KUKA KRL program: UnStackPick02.src, UnStackPick02.dat

--- UnStackPick02.src ---
&ACCESS RVP
&COMMENT UnStack Pick02
&REL 35
&PARAM EDITMASK = *
&PARAM TEMPLATE = C:\KRC\Roboter\Template\vorgabe
&PARAM DISKPATH = KRC:\R1\Program\SbtComm010Stack
DEF UnStackPick02( )
;FOLD INI;%{PE}
  ;FOLD BASISTECH INI
    GLOBAL INTERRUPT DECL 3 WHEN $STOPMESS==TRUE DO IR_STOPM ( )
    INTERRUPT ON 3
    BAS (#INITMOV,0 )
  ;ENDFOLD (BASISTECH INI)
  ;FOLD USER INI
    ;Make your modifications here

  ;ENDFOLD (USER INI)
;ENDFOLD (INI)
;FOLD COPY DATA
XPickPos = Comm010CopyTable.PickPos
;ENDFOLD
;FOLD Basic.Frame OUT Frame Dir: PickPosOfsUp, IN x: 0, IN y: 0, IN z: -150, IN a: 0 deg, IN b: 0 deg, IN c: 0 deg ;%{PE}
PickPosOfsUp = set_frame_(0, 0, -150, 0, 0, 0)
;ENDFOLD
;FOLD Basic.Frame OUT Frame Dir: PickPosOfsRUp, IN x: 0, IN y: 0, IN z: -150, IN a: 0 deg, IN b: 0 deg, IN c: 0 deg ;%{PE}
PickPosOfsRUp = set_frame_(0, 0, -150, 0, 0, 0)
;ENDFOLD
;FOLD Basic.ToolOffset IN Source Point Dir: PickPos, IN Offs Dir: PickPosOfsUp, OUT Offset Point Dir: PickPosUp ;%{PE}
XPickPosUp = tool_offs_byframe_(XPickPos, PickPosOfsUp)
;ENDFOLD
;FOLD Basic.ToolOffset IN Source Point Dir: PickPos, IN Offs Dir: PickPosOfsRUp, OUT Offset Point Dir: PickPosRUp ;%{PE}
XPickPosRUp = tool_offs_byframe_(XPickPos, PickPosOfsRUp)
;ENDFOLD
;FOLD SLIN PickPosUp CONT Vel=2 m/s CPDAT1 Tool[1] Base[0] ;%{PE}
;FOLD Parameters ;%{h}
;Params IlfProvider=kukaroboter.basistech.inlineforms.movement.spline; Kuka.IsGlobalPoint=False; Kuka.PointName=PickPosUp; Kuka.BlendingEnabled=True; Kuka.MoveDataName=CPDAT1; Kuka.VelocityPath=2; Kuka.VelocityFieldEnabled=True; Kuka.ColDetectFieldEnabled=True; Kuka.CurrentCDSetIndex=0; Kuka.MovementParameterFieldEnabled=True; IlfCommand=SLIN
;ENDFOLD
SLIN XPickPosUp WITH $VEL = SVEL_CP(2.0, , LCPDAT1), $TOOL = STOOL2(FPickPosUp), $BASE = SBASE(FPickPosUp.BASE_NO), $IPO_MODE = SIPO_MODE(FPickPosUp.IPO_FRAME), $LOAD = SLOAD(FPickPosUp.TOOL_NO), $ACC = SACC_CP(LCPDAT1), $ORI_TYPE = SORI_TYP(LCPDAT1), $APO = SAPO(LCPDAT1), $JERK = SJERK(LCPDAT1), $COLLMON_TOL_PRO[1] = USE_CM_PRO_VALUES(0) C_Spl
;ENDFOLD
;FOLD SLIN PickPos Vel=0.8 m/s CPDAT2 Tool[1] Base[0] ;%{PE}
;FOLD Parameters ;%{h}
;Params IlfProvider=kukaroboter.basistech.inlineforms.movement.spline; Kuka.IsGlobalPoint=False; Kuka.PointName=PickPos; Kuka.BlendingEnabled=False; Kuka.MoveDataName=CPDAT2; Kuka.VelocityPath=0.8; Kuka.VelocityFieldEnabled=True; Kuka.ColDetectFieldEnabled=True; Kuka.CurrentCDSetIndex=0; Kuka.MovementParameterFieldEnabled=True; IlfCommand=SLIN
;ENDFOLD
SLIN XPickPos WITH $VEL = SVEL_CP(0.8, , LCPDAT2), $TOOL = STOOL2(FPickPos), $BASE = SBASE(FPickPos.BASE_NO), $IPO_MODE = SIPO_MODE(FPickPos.IPO_FRAME), $LOAD = SLOAD(FPickPos.TOOL_NO), $ACC = SACC_CP(LCPDAT2), $ORI_TYPE = SORI_TYP(LCPDAT2), $APO = SAPO(LCPDAT2), $JERK = SJERK(LCPDAT2), $COLLMON_TOL_PRO[1] = USE_CM_PRO_VALUES(0)
;ENDFOLD
;Tool ON
;FOLD SLIN PickPosRUp CONT Vel=2 m/s CPDAT3 Tool[1] Base[0] ;%{PE}
;FOLD Parameters ;%{h}
;Params IlfProvider=kukaroboter.basistech.inlineforms.movement.spline; Kuka.IsGlobalPoint=False; Kuka.PointName=PickPosRUp; Kuka.BlendingEnabled=True; Kuka.MoveDataName=CPDAT3; Kuka.VelocityPath=2; Kuka.VelocityFieldEnabled=True; Kuka.ColDetectFieldEnabled=True; Kuka.CurrentCDSetIndex=0; Kuka.MovementParameterFieldEnabled=True; IlfCommand=SLIN
;ENDFOLD
SLIN XPickPosRUp WITH $VEL = SVEL_CP(2.0, , LCPDAT3), $TOOL = STOOL2(FPickPosRUp), $BASE = SBASE(FPickPosRUp.BASE_NO), $IPO_MODE = SIPO_MODE(FPickPosRUp.IPO_FRAME), $LOAD = SLOAD(FPickPosRUp.TOOL_NO), $ACC = SACC_CP(LCPDAT3), $ORI_TYPE = SORI_TYP(LCPDAT3), $APO = SAPO(LCPDAT3), $JERK = SJERK(LCPDAT3), $COLLMON_TOL_PRO[1] = USE_CM_PRO_VALUES(0) C_Spl
;ENDFOLD
;FOLD SbtComm010.AreaFeek IN PATH: 0, IN DELAY: 12, IN Area: 2 ;%{PE}
TRIGGER WHEN PATH=0 DELAY=12 DO ProcessComm010AreaFeek(2) PRIO = -1
;ENDFOLD
;FOLD SPTP P10 CONT Vel=100 % PDAT1 Tool[1] Base[0] ;%{PE}
;FOLD Parameters ;%{h}
;Params IlfProvider=kukaroboter.basistech.inlineforms.movement.spline; Kuka.IsGlobalPoint=False; Kuka.PointName=P10; Kuka.BlendingEnabled=True; Kuka.MoveDataPtpName=PDAT1; Kuka.VelocityPtp=100; Kuka.VelocityFieldEnabled=True; Kuka.ColDetectFieldEnabled=True; Kuka.CurrentCDSetIndex=0; Kuka.MovementParameterFieldEnabled=True; IlfCommand=SPTP
;ENDFOLD
SPTP XP10 WITH $VEL_AXIS[1] = SVEL_JOINT(100.0), $TOOL = STOOL2(FP10), $BASE = SBASE(FP10.BASE_NO), $IPO_MODE = SIPO_MODE(FP10.IPO_FRAME), $LOAD = SLOAD(FP10.TOOL_NO), $ACC_AXIS[1] = SACC_JOINT(PPDAT1), $APO = SAPO_PTP(PPDAT1), $GEAR_JERK[1] = SGEAR_JERK(PPDAT1), $COLLMON_TOL_PRO[1] = USE_CM_PRO_VALUES(0) C_Spl
;ENDFOLD
END

--- UnStackPick02.dat ---
&ACCESS RVP
&REL 35
&PARAM EDITMASK = *
&PARAM TEMPLATE = C:\KRC\Roboter\Template\vorgabe
&PARAM DISKPATH = KRC:\R1\Program\SbtComm010Stack
DEFDAT  UNSTACKPICK02
;FOLD EXTERNAL DECLARATIONS;%{PE}%MKUKATPBASIS,%CEXT,%VCOMMON,%P
;FOLD BASISTECH EXT;%{PE}%MKUKATPBASIS,%CEXT,%VEXT,%P
EXT  BAS (BAS_COMMAND  :IN,REAL  :IN )
DECL INT SUCCESS
;ENDFOLD (BASISTECH EXT)
;FOLD USER EXT;%{E}%MKUKATPUSER,%CEXT,%VEXT,%P
;Make your modifications here

;ENDFOLD (USER EXT)
;ENDFOLD (EXTERNAL DECLARATIONS)
DECL FRAME PickPosOfsUp={X 0.0,Y 0.0,Z -150.000,A 0.0,B 0.0,C 0.0}
DECL MODULEPARAM_T LAST_TP_PARAMS={PARAMS[] "BASIC.FRAMENAME=PickPosOfsRUp; BASIC.X_=0; BASIC.Y_=0; BASIC.Z_=-150; BASIC.A_=0; BASIC.B_=0; BASIC.C_=0; Kuka.VelocityFieldEnabled=True; Kuka.ColDetectFieldEnabled=True; Kuka.MovementParameterFieldEnabled=True; Kuka.IsAngleEnabled=False; Kuka.PointName=PickPos; Kuka.FrameData.base_no=0; Kuka.FrameData.tool_no=1; Kuka.FrameData.ipo_frame=#BASE; Kuka.isglobalpoint=False; Kuka.MoveDataName=CPDAT2; Kuka.MovementData.apo_fac=50; Kuka.MovementData.apo_dist=500; Kuka.MovementData.axis_acc=100; Kuka.MovementData.axis_vel=100; Kuka.MovementData.circ_typ=#BASE; Kuka.MovementData.jerk_fac=50; Kuka.MovementData.ori_typ=#VAR; Kuka.MovementData.vel=0.8; Kuka.MovementData.acc=100; Kuka.MovementData.gear_jerk=100; Kuka.MovementData.exax_ign=0; Kuka.VelocityPath=0.8; Kuka.BlendingEnabled=False; Kuka.CurrentCDSetIndex=0; Kuka.MoveDataPtpName=PDAT2; Kuka.MovementDataPdat.apo_mode=#CDIS; Kuka.MovementDataPdat.apo_dist=500; Kuka.VelocityPtp=100; SBTCOMM010.DELAYPATH=0; SBTCOMM010.DELAYTIME=12; SBTCOMM010.COMM010AREAID=2; BASIC.SOURCENAME=PickPos; BASIC.OFFSFRAME=PickPosOfsRUp; BASIC.OFFSETNAME=PickPosRUp; Kuka.FrameData.point2=           "}
DECL FRAME PickPosOfsRUp={X 0.0,Y 0.0,Z -150.000,A 0.0,B 0.0,C 0.0}
DECL E6POS XPickPosUp={X 1039.81262,Y 958.867615,Z 1330.27136,A -10.0759478,B 44.8222694,C 10.1836233,S 2,T 35,E1 0.0,E2 0.0,E3 0.0,E4 0.0,E5 0.0,E6 0.0}
DECL FDAT FPickPosUp={TOOL_NO 1,BASE_NO 0,IPO_FRAME #BASE,POINT2[] " "}
DECL LDAT LCPDAT1={VEL 2.00000,ACC 100.000,APO_DIST 500.000,APO_FAC 50.0000,AXIS_VEL 100.000,AXIS_ACC 100.000,ORI_TYP #VAR,CIRC_TYP #BASE,JERK_FAC 50.0000,GEAR_JERK 100.000,EXAX_IGN 0}
DECL E6POS XPickPos={X 1137.63843,Y 914.548584,Z 1434.98975,A -10.0759478,B 44.8222694,C 10.1836233,S 2,T 35,E1 0.0,E2 0.0,E3 0.0,E4 0.0,E5 0.0,E6 0.0}
DECL FDAT FPickPos={TOOL_NO 1,BASE_NO 0,IPO_FRAME #BASE,POINT2[] " "}
DECL LDAT LCPDAT2={VEL 0.800000,ACC 100.000,APO_DIST 500.000,APO_FAC 50.0000,AXIS_VEL 100.000,AXIS_ACC 100.000,ORI_TYP #VAR,CIRC_TYP #BASE,JERK_FAC 50.0000,GEAR_JERK 100.000,EXAX_IGN 0}
DECL E6POS XPickPosRUp={X 1039.81262,Y 958.867615,Z 1330.27136,A -10.0759478,B 44.8222694,C 10.1836233,S 2,T 35,E1 0.0,E2 0.0,E3 0.0,E4 0.0,E5 0.0,E6 0.0}
DECL FDAT FPickPosRUp={TOOL_NO 1,BASE_NO 0,IPO_FRAME #BASE,POINT2[] " "}
DECL LDAT LCPDAT3={VEL 2.00000,ACC 100.000,APO_DIST 500.000,APO_FAC 50.0000,AXIS_VEL 100.000,AXIS_ACC 100.000,ORI_TYP #VAR,CIRC_TYP #BASE,JERK_FAC 50.0000,GEAR_JERK 100.000,EXAX_IGN 0}
DECL E6POS XP10={X 2115.18164,Y 1471.05371,Z 1477.75098,A -140.399979,B 82.3619919,C -92.7671890,S 2,T 35,E1 0.0,E2 0.0,E3 0.0,E4 0.0,E5 0.0,E6 0.0}
DECL FDAT FP10={TOOL_NO 1,BASE_NO 0,IPO_FRAME #BASE,POINT2[] " "}
DECL PDAT PPDAT1={VEL 100.000,ACC 100.000,APO_DIST 500.000,APO_MODE #CDIS,GEAR_JERK 100.000,EXAX_IGN 0}
DECL PDAT PPDAT2={VEL 100.000,ACC 100.000,APO_DIST 500.000,APO_MODE #CDIS,GEAR_JERK 100.000,EXAX_IGN 0}
DECL E6POS XP9={X 1644.44800,Y 1816.82825,Z 1765.35327,A 0.0,B 89.9999924,C 34.3530197,S 2,T 35,E1 0.0,E2 0.0,E3 0.0,E4 0.0,E5 0.0,E6 0.0}
DECL FDAT FP9={TOOL_NO 1,BASE_NO 0,IPO_FRAME #BASE,POINT2[] " "}
ENDDAT
